TYPE Vec5di : ARRAY[1..5] OF DINT; END_TYPE

(* stored: Version 1.1.0.1, ProductVersion 3.1.4024.11
   DUT Vec5di: Id {afcfe2c5-a036-41f4-a52b-82b2afbc98f4} *)
